FUNCTION_BLOCK MULTIPLOTTER (* Graph image generator that allows to place 8 graphs on 1 image *)
  (* Version 1.0, AN, SWDC RTSoft *)
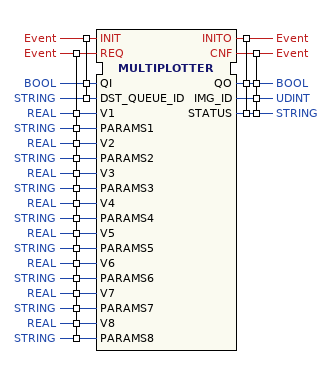
  EVENT_INPUT
    INIT WITH QI, DST_QUEUE_ID;
    REQ WITH V1, PARAMS1, V2, PARAMS2, V3, PARAMS3, V4, PARAMS4, V5, PARAMS5, V6, PARAMS6, V7, PARAMS7, V8, PARAMS8;
  END_EVENT
  EVENT_OUTPUT
    INITO WITH QO, STATUS;
    CNF WITH QO, IMG_ID, STATUS;
  END_EVENT
  VAR_INPUT
    QI : BOOL;
    DST_QUEUE_ID : STRING;
    V1 : REAL;
    PARAMS1 : STRING;
    V2 : REAL;
    PARAMS2 : STRING;
    V3 : REAL;
    PARAMS3 : STRING;
    V4 : REAL;
    PARAMS4 : STRING;
    V5 : REAL;
    PARAMS5 : STRING;
    V6 : REAL;
    PARAMS6 : STRING;
    V7 : REAL;
    PARAMS7 : STRING;
    V8 : REAL;
    PARAMS8 : STRING;
  END_VAR
  VAR_OUTPUT
    QO : BOOL;
    IMG_ID : UDINT;
    STATUS : STRING;
  END_VAR
END_FUNCTION_BLOCK
